INTERFACE iTwoDirectionalMotor // Two directional motor control

METHOD CmdRunCCW : BOOL
VAR_INPUT
END_VAR
END_METHOD

METHOD CmdRunCW : BOOL
VAR_INPUT
END_VAR
END_METHOD

METHOD Init : BOOL
VAR_INPUT
	// Message location data
	nId				: UINT ; // Identification number of object
	nParentId		: UDINT ; // Id of higher level If aplicable (0 = no parent)
END_VAR
END_METHOD

END_INTERFACE

(* stored: Version 1.1.0.1, ProductVersion 3.1.4024.11
   Itf iTwoDirectionalMotor: Id {d32567da-a499-03f5-0571-61631b1f1071}
   Method CmdRunCCW: Id {c8d703ed-592e-0314-2c47-a332655716e1}
   Method CmdRunCW: Id {f4cd52f4-5ff7-03f9-16ba-bfa76a95a3e0}
   Method Init: Id {166128ac-fa2c-0a53-3c23-eef4d035d13b} *)
